{attribute 'linkalways'} 
{attribute 'no_explicit_call' := 'This FB is a CLASS and must be accessed using methods or properties'}
{attribute 'enable_dynamic_creation'}
FUNCTION_BLOCK Node_F_VN_GetAt_TcVnRotatedRectangle EXTENDS VisionNode
VAR
    ipContainer : _ITcVnContainer;
    stElement : _TcVnRotatedRectangle;
    nIndex : _ULINT(0);
    hrPrev : _HRESULT(S_OK);
    hresult : _HRESULT(S_OK);
END_VAR

METHOD PUBLIC  Clone : I_Node
VAR
	pNode : POINTER TO Node_F_VN_GetAt_TcVnRotatedRectangle;
END_VAR
pNode := __NEW(Node_F_VN_GetAt_TcVnRotatedRectangle);
Clone := pNode^;
END_METHOD

METHOD FB_init : BOOL
VAR_INPUT
	bInitRetains : BOOL; // if TRUE, the retain variables are initialized (warm start / cold start)
	bInCopyCode : BOOL;  // if TRUE, the instance afterwards gets moved into the copy code (online change)
END_VAR
AddInput('ipContainer', ipContainer);
AddParameter('nIndex', nIndex);
AddInput('hrPrev', hrPrev);
AddOutput('stElement', stElement);
AddOutput('hresult',hresult);
END_METHOD

METHOD PROTECTED OnExecute
hresult.Value := F_VN_GetAt_TcVnRotatedRectangle(
    ipContainer := ipContainer.Value,
    stElement := stElement.Value,
    nIndex := nIndex.Value,
    hrPrev:= hrPrev.Value);
END_METHOD

METHOD PUBLIC PreExecutionCheck
VAR_INPUT
	Check : I_PreExecutionChecks;
END_VAR
Check.IsTrue(ipContainer.IsValid, 'ipContainer must be a valid container');
Check.IsTrue(ipContainer.HasType(TC_GLOBAL_CONST_LIST.ContainerType_Vector_TcVnRotatedRectangle), 'ipContainer contains incorrect type');
END_METHOD

END_FUNCTION_BLOCK

(* stored: Version 1.1.0.1, ProductVersion 3.1.4024.15
   POU Node_F_VN_GetAt_TcVnRotatedRectangle: Id {bb0a103f-c1c9-0d70-0e89-cf8ef5db33e2}, SpecialFunc None
   Folder Constructor: Id {9056a81a-f64e-0a1c-0b32-942e35fcb209}
   Method Clone: Id {ff8578c0-892a-0189-2301-55a23c8a2eb0}
   Method FB_init: Id {fca7fe25-f6ec-0082-3420-234f68775cb8}
   Method OnExecute: Id {557531dd-76af-0fa9-1274-5e2504d7e5c3}
   Method PreExecutionCheck: Id {541cb1f6-c541-0ec3-05f5-aee64d9a8083} *)
